Universal Robots PolyScope program: ur_comm_test_pal_depal_4times.urp

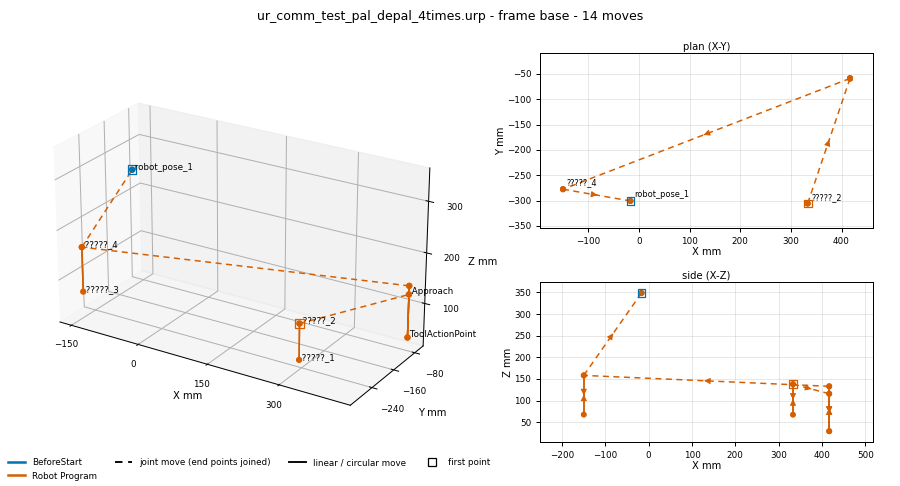
[picture p0: tool path of ur_comm_test_pal_depal_4times.urp in frame base, 14 of 14 moves have a stored position in this frame; points joined in program order, loops and branches not executed]
Program ur_comm_test_pal_depal_10times (installation=default directory=/programs/usbdisk/zivid-python-test/ur_comm_test_sample createdIn=5.5.1 lastSavedIn=5.21.0 robotSerialNumber=20195300395)
Calibrated DH parameters: a=[-0.000108, -0.14067, -0.21248, -0.000061, -0.000086, 0]; d=[0.151815, 81.30975, -77.69219, -3.486516, 0.085386, 0.091974]; alpha=[1.569683, -0.002449, 0.004563, 1.571204, -1.571811, 0]; deltaTheta=[0, -0.955759, 1.033289, -0.077525, 0.000001, 0]
InitVariablesNode variables(variable(name=Pallet_1_cnt, expression=1), variable(name=Pallet_1_cnt_1, expression=1), variable(name=Pallet_1_lct, expression=1), variable(name=Pallet_1_lct_1, expression=1), variable(name=Pallet_1_lno, expression=1), variable(name=Pallet_1_lno_1, expression=1), variable(name=Pallet_1_sep, expression=False), variable(name=Pallet_1_sep_1, expression=False), variable(name=Pallet_1_tct, expression=1), variable(name=Pallet_1_tct_1, expression=1), variable(name=qNearApproach, expression=[0,0,0,0,0,0]), variable(name=qNearApproach_1, expression=[0,0,0,0,0,0]))
BeforeStart
  Set DigitalOutput pin=conveyor_on; digitalValue=1
  count := 0
  URCap 2FG 놓기 (OnRobot, OnRobot A/S) dataModel(twofg.external-grip.target-width=0.03670000076293945, twofg.internal-grip.target-width=0.05070000076293945)
  MoveJ speed 15 deg/s, acceleration 15 deg/s^2 (useActiveTCP=true optimoveEnabled=true optiMoveSpeed=1 optiMoveAcceleration=1) feature=Base
    Waypoint robot_pose_1: TCP in base x=-16.534 y=-300.847 z=348.638 mm, rx=2.6839 ry=0.1063 rz=-0.0079 rad; joints [-46.382, -62.621, -71.979, -115.359, 73.035, -143.967] deg; TCP offset x=-7.625 y=23.932 z=143.735 mm, rx=0 ry=0 rz=0 rad
  Script: write_output_integer_register(24,count)
  Script: write_output_boolean_register(64,False)
Robot Program (runOnlyOnce=false)
  Wait Condition expression=read_input_boolean_register(125)
  count := count+1
  Script: write_output_integer_register(24,count)
  Script: write_output_boolean_register(64,True)
  Script: read_input_boolean_register(125)
  Loop Counting (count=4) loopVariable(name=루프_1)
    Loop Counting (count=6) loopVariable(name=루프_2)
      MoveJ speed 60 deg/s, acceleration 80 deg/s^2 (useActiveTCP=true optimoveEnabled=true optiMoveSpeed=1 optiMoveAcceleration=1) feature=Base
        Waypoint 웨이포인트_2: TCP in base x=333.162 y=-305.802 z=138.045 mm, rx=2.2214 ry=2.2214 rz=0 rad; joints [-26.216, -117.027, -61.814, -91.097, 90.185, -206.198] deg
      MoveL speed 250 mm/s, acceleration 1200 mm/s^2 (useActiveTCP=true optimoveEnabled=true optiMoveSpeed=1 optiMoveAcceleration=1) feature=Base
        Waypoint 웨이포인트_1: TCP in base x=333.162 y=-305.802 z=67.503 mm, rx=2.2214 ry=2.2214 rz=0 rad; joints [-26.24, -119.399, -77.36, -73.18, 90.18, -206.146] deg
        URCap 2FG 그립 (OnRobot, OnRobot A/S) dataModel(twofg.external-grip.target-width=0.02370000076293945, twofg.internal-grip.target-width=0.03770000076293945)
        Waypoint 웨이포인트_2: TCP in base x=333.162 y=-305.802 z=138.045 mm, rx=2.2214 ry=2.2214 rz=0 rad; joints [-26.216, -117.027, -61.814, -91.097, 90.185, -206.198] deg
      URCap 팔레타이징 (polyscope-pallet-impl, Universal Robots) dataModel(palletFeature=Base, isPalletizing=true, Variable(key=referencePoint, variable(featureName=referencePoint)), Variable(key=separatorPoint, variable(featureName=separatorPoint)), Variable(key=qNearApproach, variable(name=qNearApproach, initializeExpression=[0,0,0,0,0,0])), Variable(key=name, variable(name=Pallet_1)), Variable(key=globalCountingVariable, variable(name=Pallet_1_cnt, initializeExpression=1)), Variable(key=layerNumberVariable, variable(name=Pallet_1_lno, initializeExpression=1)), Variable(key=layerCountingVariable, variable(name=Pallet_1_lct, initializeExpression=1)), Variable(key=handleSeparatorVariable, variable(name=Pallet_1_sep, initializeExpression=False)), Variable(key=totalCountVariable, variable(name=Pallet_1_tct, initializeExpression=1)), Length(key=objectHeight value=0.03 unit=M)); state(isChildrenLocked=true)
        URCap 패턴 (polyscope-pallet-impl, Universal Robots) state(isChildrenLocked=true)
          URCap 패턴 (polyscope-pallet-impl, Universal Robots) dataModel(UUID=d919b560-e99a-480d-bc1f-cb570735da14, patternType=GRID, rows=3, columns=2, Variable(key=nameVariable, variable(name=Grid_Pattern_1))); state(isChildrenLocked=true)
            URCap 아이템 (polyscope-pallet-impl, Universal Robots) dataModel(UUID=ee1cad20-2e71-4b8d-ab70-a290e76e5d6c, patternType=GRID, index=0, calibrationDeltaTheta=[6.716763317901001E-8, -0.9557590612475653, 1.0332894801482315, -0.07752547289049558, 5.674308259095984E-7, -2.281062283008531E-7], calibrationA=[-1.0844059639211092E-4, -0.14067031953614179, -0.21248043873134673, -6.078177536491715E-5, -8.613979399887485E-5, 0.0], calibrationD=[0.15181475343250603, 81.30975015896925, -77.6921895952701, -3.486515920890218, 0.08538604408418736, 0.09197393797432639], calibrationAlpha=[1.569682990986815, -0.0024489725605047743, 0.004563020512108627, 1.571204384472482, -1.5718110539936228, 0.0], calibrationJointChecksum=[-1321669567, -1322594988, 822688479, -1328072335, -1327094287, -1329556568], calibrationStatus=2, calibrationValidChecksum=true, baseToFeature=[0.0, 0.0, 0.0, 0.0, 0.0, 0.0], TCPOffset=[-0.00762820289468219, 0.0239501142926695, 0.14372303756847724, -4.3315942804722315E-5, 7.042533500568108E-6, 2.3758754532917458E-5], Variable(key=variable, variable(name=CornerItem_1)), JointPositions(key=jointpositions, JointPosition(key=[1], Angle(key=pos value=0.230122 unit=RAD)), JointPosition(key=[2], Angle(key=pos value=-2.124559 unit=RAD)), JointPosition(key=[3], Angle(key=pos value=-1.476286 unit=RAD)), JointPosition(key=[4], Angle(key=pos value=-1.110532 unit=RAD)), JointPosition(key=[5], Angle(key=pos value=1.5737 unit=RAD)), JointPosition(key=[6], Angle(key=pos value=-1.360397 unit=RAD))))
            URCap 아이템 (polyscope-pallet-impl, Universal Robots) dataModel(UUID=2ec53ba5-ed44-4377-a54f-87662cf6edc9, patternType=GRID, index=1, calibrationDeltaTheta=[6.716763317901001E-8, -0.9557590612475653, 1.0332894801482315, -0.07752547289049558, 5.674308259095984E-7, -2.281062283008531E-7], calibrationA=[-1.0844059639211092E-4, -0.14067031953614179, -0.21248043873134673, -6.078177536491715E-5, -8.613979399887485E-5, 0.0], calibrationD=[0.15181475343250603, 81.30975015896925, -77.6921895952701, -3.486515920890218, 0.08538604408418736, 0.09197393797432639], calibrationAlpha=[1.569682990986815, -0.0024489725605047743, 0.004563020512108627, 1.571204384472482, -1.5718110539936228, 0.0], calibrationJointChecksum=[-1321669567, -1322594988, 822688479, -1328072335, -1327094287, -1329556568], calibrationStatus=2, calibrationValidChecksum=true, baseToFeature=[0.0, 0.0, 0.0, 0.0, 0.0, 0.0], TCPOffset=[-0.007627364228596889, 0.023926276031487913, 0.1437254493979939, 1.6298927572986975E-5, -1.936015947561922E-6, -2.0279970492899247E-5], Variable(key=variable, variable(name=CornerItem_2)), JointPositions(key=jointpositions, JointPosition(key=[1], Angle(key=pos value=0.32864 unit=RAD)), JointPosition(key=[2], Angle(key=pos value=-1.666236 unit=RAD)), JointPosition(key=[3], Angle(key=pos value=-2.130058 unit=RAD)), JointPosition(key=[4], Angle(key=pos value=-0.915088 unit=RAD)), JointPosition(key=[5], Angle(key=pos value=1.573564 unit=RAD)), JointPosition(key=[6], Angle(key=pos value=-1.259999 unit=RAD))))
            URCap 아이템 (polyscope-pallet-impl, Universal Robots) dataModel(UUID=892b0312-8469-4b11-924f-1544095aac69, patternType=GRID, index=2, calibrationDeltaTheta=[6.716763317901001E-8, -0.9557590612475653, 1.0332894801482315, -0.07752547289049558, 5.674308259095984E-7, -2.281062283008531E-7], calibrationA=[-1.0844059639211092E-4, -0.14067031953614179, -0.21248043873134673, -6.078177536491715E-5, -8.613979399887485E-5, 0.0], calibrationD=[0.15181475343250603, 81.30975015896925, -77.6921895952701, -3.486515920890218, 0.08538604408418736, 0.09197393797432639], calibrationAlpha=[1.569682990986815, -0.0024489725605047743, 0.004563020512108627, 1.571204384472482, -1.5718110539936228, 0.0], calibrationJointChecksum=[-1321669567, -1322594988, 822688479, -1328072335, -1327094287, -1329556568], calibrationStatus=2, calibrationValidChecksum=true, baseToFeature=[0.0, 0.0, 0.0, 0.0, 0.0, 0.0], TCPOffset=[-0.007639878420080737, 0.023943869668825668, 0.14373765785164358, -1.943663654326589E-5, -1.5468052752266034E-5, 3.456527941839842E-6], Variable(key=variable, variable(name=CornerItem_3)), JointPositions(key=jointpositions, JointPosition(key=[1], Angle(key=pos value=0.118809 unit=RAD)), JointPosition(key=[2], Angle(key=pos value=-1.718406 unit=RAD)), JointPosition(key=[3], Angle(key=pos value=-2.068775 unit=RAD)), JointPosition(key=[4], Angle(key=pos value=-0.924192 unit=RAD)), JointPosition(key=[5], Angle(key=pos value=1.573526 unit=RAD)), JointPosition(key=[6], Angle(key=pos value=-1.469977 unit=RAD))))
            URCap 아이템 (polyscope-pallet-impl, Universal Robots) dataModel(UUID=cf353ae9-dbdd-4e16-bdff-710f563f51b7, patternType=GRID, index=3, calibrationDeltaTheta=[6.716763317901001E-8, -0.9557590612475653, 1.0332894801482315, -0.07752547289049558, 5.674308259095984E-7, -2.281062283008531E-7], calibrationA=[-1.0844059639211092E-4, -0.14067031953614179, -0.21248043873134673, -6.078177536491715E-5, -8.613979399887485E-5, 0.0], calibrationD=[0.15181475343250603, 81.30975015896925, -77.6921895952701, -3.486515920890218, 0.08538604408418736, 0.09197393797432639], calibrationAlpha=[1.569682990986815, -0.0024489725605047743, 0.004563020512108627, 1.571204384472482, -1.5718110539936228, 0.0], calibrationJointChecksum=[-1321669567, -1322594988, 822688479, -1328072335, -1327094287, -1329556568], calibrationStatus=2, calibrationValidChecksum=true, baseToFeature=[0.0, 0.0, 0.0, 0.0, 0.0, 0.0], TCPOffset=[-0.0076283249516490015, 0.02393296756205482, 0.14376242105826337, -1.8085091406019513E-5, -4.76246665041877E-5, 1.1126998149954308E-5], Variable(key=variable, variable(name=CornerItem_4)), JointPositions(key=jointpositions, JointPosition(key=[1], Angle(key=pos value=0.080239 unit=RAD)), JointPosition(key=[2], Angle(key=pos value=-2.155316 unit=RAD)), JointPosition(key=[3], Angle(key=pos value=-1.42445 unit=RAD)), JointPosition(key=[4], Angle(key=pos value=-1.131606 unit=RAD)), JointPosition(key=[5], Angle(key=pos value=1.573688 unit=RAD)), JointPosition(key=[6], Angle(key=pos value=-1.510421 unit=RAD))))
        URCap 레이어 (polyscope-pallet-impl, Universal Robots) dataModel(separators=[false], selectedPatterns=[d919b560-e99a-480d-bc1f-cb570735da14])
        URCap 각각의 아이템 (polyscope-pallet-impl, Universal Robots) dataModel(selectedPattern=d919b560-e99a-480d-bc1f-cb570735da14, selectedPosition=ee1cad20-2e71-4b8d-ab70-a290e76e5d6c, Approach_calibrationDeltaTheta=[6.716763317901001E-8, -0.9557590612475653, 1.0332894801482315, -0.07752547289049558, 5.674308259095984E-7, -2.281062283008531E-7], Approach_calibrationA=[-1.0844059639211092E-4, -0.14067031953614179, -0.21248043873134673, -6.078177536491715E-5, -8.613979399887485E-5, 0.0], Approach_calibrationD=[0.15181475343250603, 81.30975015896925, -77.6921895952701, -3.486515920890218, 0.08538604408418736, 0.09197393797432639], Approach_calibrationAlpha=[1.569682990986815, -0.0024489725605047743, 0.004563020512108627, 1.571204384472482, -1.5718110539936228, 0.0], Approach_calibrationJointChecksum=[-1321669567, -1322594988, 822688479, -1328072335, -1327094287, -1329556568], Approach_calibrationStatus=2, Approach_calibrationValidChecksum=true, Approach_baseToFeature=[0.0, 0.0, 0.0, 0.0, 0.0, 0.0], Approach_TCPOffset=[-0.0076294742125221915, 0.02392315779155893, 0.14376079906325706, 2.9702410288334196E-5, -6.399436710385144E-5, -4.55675022656733E-5], Exit_calibrationDeltaTheta=[6.716763317901001E-8, -0.9557590612475653, 1.0332894801482315, -0.07752547289049558, 5.674308259095984E-7, -2.281062283008531E-7], Exit_calibrationA=[-1.0844059639211092E-4, -0.14067031953614179, -0.21248043873134673, -6.078177536491715E-5, -8.613979399887485E-5, 0.0], Exit_calibrationD=[0.15181475343250603, 81.30975015896925, -77.6921895952701, -3.486515920890218, 0.08538604408418736, 0.09197393797432639], Exit_calibrationAlpha=[1.569682990986815, -0.0024489725605047743, 0.004563020512108627, 1.571204384472482, -1.5718110539936228, 0.0], Exit_calibrationJointChecksum=[-1321669567, -1322594988, 822688479, -1328072335, -1327094287, -1329556568], Exit_calibrationStatus=2, Exit_calibrationValidChecksum=true, Exit_baseToFeature=[0.0, 0.0, 0.0, 0.0, 0.0, 0.0], Exit_TCPOffset=[-0.007615351300449602, 0.02389728385555888, 0.14374352147036207, 2.5680027780448787E-5, -3.149176289617292E-6, -3.7337634040478105E-5], currentWizardState=LANDING, Pose(key=refBaseToFeature, Position(key=posePosition, Length(key=X value=0 unit=M), Length(key=Y value=0 unit=M), Length(key=Z value=0 unit=M)), Rotation(key=poseRotation, Angle(key=RX value=0 unit=RAD), Angle(key=RY value=0 unit=RAD), Angle(key=RZ value=0 unit=RAD))), Pose(key=refPose, Position(key=posePosition, Length(key=X value=0.416803 unit=M), Length(key=Y value=-0.059002 unit=M), Length(key=Z value=0.029418 unit=M)), Rotation(key=poseRotation, Angle(key=RX value=3.14136 unit=RAD), Angle(key=RY value=0.034493 unit=RAD), Angle(key=RZ value=0.000012 unit=RAD))), JointPositions(key=Approach_jointpositions, JointPosition(key=[1], Angle(key=pos value=0.23048 unit=RAD)), JointPosition(key=[2], Angle(key=pos value=-2.025888 unit=RAD)), JointPosition(key=[3], Angle(key=pos value=-1.207737 unit=RAD)), JointPosition(key=[4], Angle(key=pos value=-1.477755 unit=RAD)), JointPosition(key=[5], Angle(key=pos value=1.574011 unit=RAD)), JointPosition(key=[6], Angle(key=pos value=-1.361408 unit=RAD))), JointPositions(key=Exit_jointpositions, JointPosition(key=[1], Angle(key=pos value=0.2306 unit=RAD)), JointPosition(key=[2], Angle(key=pos value=-2.021999 unit=RAD)), JointPosition(key=[3], Angle(key=pos value=-1.133203 unit=RAD)), JointPosition(key=[4], Angle(key=pos value=-1.556178 unit=RAD)), JointPosition(key=[5], Angle(key=pos value=1.574003 unit=RAD)), JointPosition(key=[6], Angle(key=pos value=-1.361636 unit=RAD))))
          URCap 생성된 이동 (polyscope-pallet-impl, Universal Robots) state(isChildrenLocked=true)
            MoveJ speed 60 deg/s, acceleration 80 deg/s^2 (useActiveTCP=true optimoveEnabled=true optiMoveSpeed=1 optiMoveAcceleration=1) feature=referencePoint
              Waypoint Approach: TCP in base x=416.798 y=-58.994 z=115.935 mm, rx=3.1414 ry=0.0346 rz=-0.0001 rad; joints [13.206, -116.075, -69.198, -84.669, 90.184, -78.003] deg; TCP offset x=-7.629 y=23.923 z=143.761 mm, rx=0 ry=-0.0001 rz=0 rad; feature pose in base x=416.803 y=-59.002 z=29.418 mm, rx=3.1414 ry=0.0345 rz=0 rad
            MoveL speed 250 mm/s, acceleration 1200 mm/s^2 (useActiveTCP=true optimoveEnabled=true optiMoveSpeed=1 optiMoveAcceleration=1) feature(featureName=referencePoint)
              Waypoint ToolActionPoint: TCP in base x=416.803 y=-59.002 z=29.418 mm, rx=3.1414 ry=0.0345 rz=0 rad; joints [13.185, -121.728, -84.585, -63.629, 90.166, -77.945] deg; TCP offset x=-7.628 y=23.95 z=143.723 mm, rx=0 ry=0 rz=0 rad
            Folder Tool action
              URCap 2FG 놓기 (OnRobot, OnRobot A/S) dataModel(twofg.external-grip.target-width=0.03670000076293945, twofg.internal-grip.target-width=0.05070000076293945)
            MoveL speed 250 mm/s, acceleration 1200 mm/s^2 (useActiveTCP=true optimoveEnabled=true optiMoveSpeed=1 optiMoveAcceleration=1) feature(featureName=referencePoint)
              Waypoint Exit: TCP in base x=416.812 y=-58.968 z=133.052 mm, rx=3.1414 ry=0.0346 rz=0 rad; joints [13.212, -115.852, -64.928, -89.162, 90.184, -78.016] deg; TCP offset x=-7.615 y=23.897 z=143.744 mm, rx=0 ry=0 rz=0 rad
    Loop Counting (count=6) loopVariable(name=루프_3)
      URCap 팔레타이징 (polyscope-pallet-impl, Universal Robots) dataModel(palletFeature=Base, isPalletizing=false, Length(key=objectHeight value=0.03 unit=M), Variable(key=referencePoint, variable(featureName=referencePoin_1)), Variable(key=separatorPoint, variable(featureName=separatorPoin_1)), Variable(key=qNearApproach, variable(name=qNearApproach_1, initializeExpression=[0,0,0,0,0,0])), Variable(key=name, variable(name=Pallet_2)), Variable(key=globalCountingVariable, variable(name=Pallet_1_cnt_1, initializeExpression=1)), Variable(key=layerCountingVariable, variable(name=Pallet_1_lct_1, initializeExpression=1)), Variable(key=layerNumberVariable, variable(name=Pallet_1_lno_1, initializeExpression=1)), Variable(key=handleSeparatorVariable, variable(name=Pallet_1_sep_1, initializeExpression=False)), Variable(key=totalCountVariable, variable(name=Pallet_1_tct_1, initializeExpression=1))); state(isChildrenLocked=true)
        URCap 패턴 (polyscope-pallet-impl, Universal Robots) state(isChildrenLocked=true)
          URCap 패턴 (polyscope-pallet-impl, Universal Robots) dataModel(UUID=d919b560-e99a-480d-bc1f-cb570735da14, patternType=GRID, rows=3, columns=2, Variable(key=nameVariable, variable(name=Grid_Pattern_2))); state(isChildrenLocked=true)
            URCap 아이템 (polyscope-pallet-impl, Universal Robots) dataModel(UUID=ee1cad20-2e71-4b8d-ab70-a290e76e5d6c, patternType=GRID, index=0, calibrationDeltaTheta=[6.716763317901001E-8, -0.9557590612475653, 1.0332894801482315, -0.07752547289049558, 5.674308259095984E-7, -2.281062283008531E-7], calibrationA=[-1.0844059639211092E-4, -0.14067031953614179, -0.21248043873134673, -6.078177536491715E-5, -8.613979399887485E-5, 0.0], calibrationD=[0.15181475343250603, 81.30975015896925, -77.6921895952701, -3.486515920890218, 0.08538604408418736, 0.09197393797432639], calibrationAlpha=[1.569682990986815, -0.0024489725605047743, 0.004563020512108627, 1.571204384472482, -1.5718110539936228, 0.0], calibrationJointChecksum=[-1321669567, -1322594988, 822688479, -1328072335, -1327094287, -1329556568], calibrationStatus=2, calibrationValidChecksum=true, baseToFeature=[0.0, 0.0, 0.0, 0.0, 0.0, 0.0], TCPOffset=[-0.00762820289468219, 0.0239501142926695, 0.14372303756847724, -4.3315942804722315E-5, 7.042533500568108E-6, 2.3758754532917458E-5], JointPositions(key=jointpositions, JointPosition(key=[1], Angle(key=pos value=0.230122 unit=RAD)), JointPosition(key=[2], Angle(key=pos value=-2.124559 unit=RAD)), JointPosition(key=[3], Angle(key=pos value=-1.476286 unit=RAD)), JointPosition(key=[4], Angle(key=pos value=-1.110532 unit=RAD)), JointPosition(key=[5], Angle(key=pos value=1.5737 unit=RAD)), JointPosition(key=[6], Angle(key=pos value=-1.360397 unit=RAD))), Variable(key=variable, variable(name=CornerItem_5)))
            URCap 아이템 (polyscope-pallet-impl, Universal Robots) dataModel(UUID=2ec53ba5-ed44-4377-a54f-87662cf6edc9, patternType=GRID, index=1, calibrationDeltaTheta=[6.716763317901001E-8, -0.9557590612475653, 1.0332894801482315, -0.07752547289049558, 5.674308259095984E-7, -2.281062283008531E-7], calibrationA=[-1.0844059639211092E-4, -0.14067031953614179, -0.21248043873134673, -6.078177536491715E-5, -8.613979399887485E-5, 0.0], calibrationD=[0.15181475343250603, 81.30975015896925, -77.6921895952701, -3.486515920890218, 0.08538604408418736, 0.09197393797432639], calibrationAlpha=[1.569682990986815, -0.0024489725605047743, 0.004563020512108627, 1.571204384472482, -1.5718110539936228, 0.0], calibrationJointChecksum=[-1321669567, -1322594988, 822688479, -1328072335, -1327094287, -1329556568], calibrationStatus=2, calibrationValidChecksum=true, baseToFeature=[0.0, 0.0, 0.0, 0.0, 0.0, 0.0], TCPOffset=[-0.007627364228596889, 0.023926276031487913, 0.1437254493979939, 1.6298927572986975E-5, -1.936015947561922E-6, -2.0279970492899247E-5], JointPositions(key=jointpositions, JointPosition(key=[1], Angle(key=pos value=0.32864 unit=RAD)), JointPosition(key=[2], Angle(key=pos value=-1.666236 unit=RAD)), JointPosition(key=[3], Angle(key=pos value=-2.130058 unit=RAD)), JointPosition(key=[4], Angle(key=pos value=-0.915088 unit=RAD)), JointPosition(key=[5], Angle(key=pos value=1.573564 unit=RAD)), JointPosition(key=[6], Angle(key=pos value=-1.259999 unit=RAD))), Variable(key=variable, variable(name=CornerItem_6)))
            URCap 아이템 (polyscope-pallet-impl, Universal Robots) dataModel(UUID=892b0312-8469-4b11-924f-1544095aac69, patternType=GRID, index=2, calibrationDeltaTheta=[6.716763317901001E-8, -0.9557590612475653, 1.0332894801482315, -0.07752547289049558, 5.674308259095984E-7, -2.281062283008531E-7], calibrationA=[-1.0844059639211092E-4, -0.14067031953614179, -0.21248043873134673, -6.078177536491715E-5, -8.613979399887485E-5, 0.0], calibrationD=[0.15181475343250603, 81.30975015896925, -77.6921895952701, -3.486515920890218, 0.08538604408418736, 0.09197393797432639], calibrationAlpha=[1.569682990986815, -0.0024489725605047743, 0.004563020512108627, 1.571204384472482, -1.5718110539936228, 0.0], calibrationJointChecksum=[-1321669567, -1322594988, 822688479, -1328072335, -1327094287, -1329556568], calibrationStatus=2, calibrationValidChecksum=true, baseToFeature=[0.0, 0.0, 0.0, 0.0, 0.0, 0.0], TCPOffset=[-0.007639878420080737, 0.023943869668825668, 0.14373765785164358, -1.943663654326589E-5, -1.5468052752266034E-5, 3.456527941839842E-6], JointPositions(key=jointpositions, JointPosition(key=[1], Angle(key=pos value=0.118809 unit=RAD)), JointPosition(key=[2], Angle(key=pos value=-1.718406 unit=RAD)), JointPosition(key=[3], Angle(key=pos value=-2.068775 unit=RAD)), JointPosition(key=[4], Angle(key=pos value=-0.924192 unit=RAD)), JointPosition(key=[5], Angle(key=pos value=1.573526 unit=RAD)), JointPosition(key=[6], Angle(key=pos value=-1.469977 unit=RAD))), Variable(key=variable, variable(name=CornerItem_7)))
            URCap 아이템 (polyscope-pallet-impl, Universal Robots) dataModel(UUID=cf353ae9-dbdd-4e16-bdff-710f563f51b7, patternType=GRID, index=3, calibrationDeltaTheta=[6.716763317901001E-8, -0.9557590612475653, 1.0332894801482315, -0.07752547289049558, 5.674308259095984E-7, -2.281062283008531E-7], calibrationA=[-1.0844059639211092E-4, -0.14067031953614179, -0.21248043873134673, -6.078177536491715E-5, -8.613979399887485E-5, 0.0], calibrationD=[0.15181475343250603, 81.30975015896925, -77.6921895952701, -3.486515920890218, 0.08538604408418736, 0.09197393797432639], calibrationAlpha=[1.569682990986815, -0.0024489725605047743, 0.004563020512108627, 1.571204384472482, -1.5718110539936228, 0.0], calibrationJointChecksum=[-1321669567, -1322594988, 822688479, -1328072335, -1327094287, -1329556568], calibrationStatus=2, calibrationValidChecksum=true, baseToFeature=[0.0, 0.0, 0.0, 0.0, 0.0, 0.0], TCPOffset=[-0.0076283249516490015, 0.02393296756205482, 0.14376242105826337, -1.8085091406019513E-5, -4.76246665041877E-5, 1.1126998149954308E-5], JointPositions(key=jointpositions, JointPosition(key=[1], Angle(key=pos value=0.080239 unit=RAD)), JointPosition(key=[2], Angle(key=pos value=-2.155316 unit=RAD)), JointPosition(key=[3], Angle(key=pos value=-1.42445 unit=RAD)), JointPosition(key=[4], Angle(key=pos value=-1.131606 unit=RAD)), JointPosition(key=[5], Angle(key=pos value=1.573688 unit=RAD)), JointPosition(key=[6], Angle(key=pos value=-1.510421 unit=RAD))), Variable(key=variable, variable(name=CornerItem_8)))
        URCap 레이어 (polyscope-pallet-impl, Universal Robots) dataModel(separators=[false], selectedPatterns=[d919b560-e99a-480d-bc1f-cb570735da14])
        URCap 각각의 아이템 (polyscope-pallet-impl, Universal Robots) dataModel(selectedPattern=d919b560-e99a-480d-bc1f-cb570735da14, selectedPosition=ee1cad20-2e71-4b8d-ab70-a290e76e5d6c, Approach_calibrationDeltaTheta=[6.716763317901001E-8, -0.9557590612475653, 1.0332894801482315, -0.07752547289049558, 5.674308259095984E-7, -2.281062283008531E-7], Approach_calibrationA=[-1.0844059639211092E-4, -0.14067031953614179, -0.21248043873134673, -6.078177536491715E-5, -8.613979399887485E-5, 0.0], Approach_calibrationD=[0.15181475343250603, 81.30975015896925, -77.6921895952701, -3.486515920890218, 0.08538604408418736, 0.09197393797432639], Approach_calibrationAlpha=[1.569682990986815, -0.0024489725605047743, 0.004563020512108627, 1.571204384472482, -1.5718110539936228, 0.0], Approach_calibrationJointChecksum=[-1321669567, -1322594988, 822688479, -1328072335, -1327094287, -1329556568], Approach_calibrationStatus=2, Approach_calibrationValidChecksum=true, Approach_baseToFeature=[0.0, 0.0, 0.0, 0.0, 0.0, 0.0], Approach_TCPOffset=[-0.0076294742125221915, 0.02392315779155893, 0.14376079906325706, 2.9702410288334196E-5, -6.399436710385144E-5, -4.55675022656733E-5], Exit_calibrationDeltaTheta=[6.716763317901001E-8, -0.9557590612475653, 1.0332894801482315, -0.07752547289049558, 5.674308259095984E-7, -2.281062283008531E-7], Exit_calibrationA=[-1.0844059639211092E-4, -0.14067031953614179, -0.21248043873134673, -6.078177536491715E-5, -8.613979399887485E-5, 0.0], Exit_calibrationD=[0.15181475343250603, 81.30975015896925, -77.6921895952701, -3.486515920890218, 0.08538604408418736, 0.09197393797432639], Exit_calibrationAlpha=[1.569682990986815, -0.0024489725605047743, 0.004563020512108627, 1.571204384472482, -1.5718110539936228, 0.0], Exit_calibrationJointChecksum=[-1321669567, -1322594988, 822688479, -1328072335, -1327094287, -1329556568], Exit_calibrationStatus=2, Exit_calibrationValidChecksum=true, Exit_baseToFeature=[0.0, 0.0, 0.0, 0.0, 0.0, 0.0], Exit_TCPOffset=[-0.007615351300449602, 0.02389728385555888, 0.14374352147036207, 2.5680027780448787E-5, -3.149176289617292E-6, -3.7337634040478105E-5], currentWizardState=LANDING, Pose(key=refBaseToFeature, Position(key=posePosition, Length(key=X value=0 unit=M), Length(key=Y value=0 unit=M), Length(key=Z value=0 unit=M)), Rotation(key=poseRotation, Angle(key=RX value=0 unit=RAD), Angle(key=RY value=0 unit=RAD), Angle(key=RZ value=0 unit=RAD))), Pose(key=refPose, Position(key=posePosition, Length(key=X value=0.416803 unit=M), Length(key=Y value=-0.059002 unit=M), Length(key=Z value=0.029418 unit=M)), Rotation(key=poseRotation, Angle(key=RX value=3.14136 unit=RAD), Angle(key=RY value=0.034493 unit=RAD), Angle(key=RZ value=0.000012 unit=RAD))), JointPositions(key=Approach_jointpositions, JointPosition(key=[1], Angle(key=pos value=0.23048 unit=RAD)), JointPosition(key=[2], Angle(key=pos value=-2.025888 unit=RAD)), JointPosition(key=[3], Angle(key=pos value=-1.207737 unit=RAD)), JointPosition(key=[4], Angle(key=pos value=-1.477755 unit=RAD)), JointPosition(key=[5], Angle(key=pos value=1.574011 unit=RAD)), JointPosition(key=[6], Angle(key=pos value=-1.361408 unit=RAD))), JointPositions(key=Exit_jointpositions, JointPosition(key=[1], Angle(key=pos value=0.2306 unit=RAD)), JointPosition(key=[2], Angle(key=pos value=-2.021999 unit=RAD)), JointPosition(key=[3], Angle(key=pos value=-1.133203 unit=RAD)), JointPosition(key=[4], Angle(key=pos value=-1.556178 unit=RAD)), JointPosition(key=[5], Angle(key=pos value=1.574003 unit=RAD)), JointPosition(key=[6], Angle(key=pos value=-1.361636 unit=RAD))))
          URCap 생성된 이동 (polyscope-pallet-impl, Universal Robots) state(isChildrenLocked=true)
            MoveJ speed 60 deg/s, acceleration 80 deg/s^2 (useActiveTCP=true optimoveEnabled=true optiMoveSpeed=1 optiMoveAcceleration=1) feature=referencePoin_1
              Waypoint Approach: TCP in base x=416.798 y=-58.994 z=115.935 mm, rx=3.1414 ry=0.0346 rz=-0.0001 rad; joints [13.206, -116.075, -69.198, -84.669, 90.184, -78.003] deg; TCP offset x=-7.629 y=23.923 z=143.761 mm, rx=0 ry=-0.0001 rz=0 rad
            MoveL speed 250 mm/s, acceleration 1200 mm/s^2 (useActiveTCP=true optimoveEnabled=true optiMoveSpeed=1 optiMoveAcceleration=1) feature(featureName=referencePoin_1)
              Waypoint ToolActionPoint: TCP in base x=416.803 y=-59.002 z=29.418 mm, rx=3.1414 ry=0.0345 rz=0 rad; joints [13.185, -121.728, -84.585, -63.629, 90.166, -77.945] deg; TCP offset x=-7.628 y=23.95 z=143.723 mm, rx=0 ry=0 rz=0 rad
            Folder Tool action
              URCap 2FG 그립 (OnRobot, OnRobot A/S) dataModel(twofg.external-grip.target-width=0.02370000076293945, twofg.internal-grip.target-width=0.03770000076293945)
            MoveL speed 250 mm/s, acceleration 1200 mm/s^2 (useActiveTCP=true optimoveEnabled=true optiMoveSpeed=1 optiMoveAcceleration=1) feature(featureName=referencePoin_1)
              Waypoint Exit: TCP in base x=416.812 y=-58.968 z=133.052 mm, rx=3.1414 ry=0.0346 rz=0 rad; joints [13.212, -115.852, -64.928, -89.162, 90.184, -78.016] deg; TCP offset x=-7.615 y=23.897 z=143.744 mm, rx=0 ry=0 rz=0 rad
      MoveJ speed 60 deg/s, acceleration 80 deg/s^2 (useActiveTCP=true optimoveEnabled=true optiMoveSpeed=1 optiMoveAcceleration=1) feature=Base
        Waypoint 웨이포인트_4: TCP in base x=-149.78 y=-277.687 z=158.255 mm, rx=-2.191 ry=2.2515 rz=0 rad; joints [-89.108, -86.57, -93.896, -89.476, 90.215, -87.455] deg; TCP offset x=-7.625 y=23.932 z=143.735 mm, rx=0 ry=0 rz=0 rad
      MoveL speed 250 mm/s, acceleration 1200 mm/s^2 (useActiveTCP=true optimoveEnabled=true optiMoveSpeed=1 optiMoveAcceleration=1) feature=Base
        Waypoint 웨이포인트_3: TCP in base x=-149.78 y=-277.687 z=67.712 mm, rx=-2.191 ry=2.2515 rz=0 rad; joints [-89.143, -91.506, -114.239, -64.197, 90.191, -87.387] deg
        URCap 2FG 놓기 (OnRobot, OnRobot A/S) dataModel(twofg.external-grip.target-width=0.03670000076293945, twofg.internal-grip.target-width=0.05070000076293945)
        Waypoint 웨이포인트_4: TCP in base x=-149.78 y=-277.687 z=158.255 mm, rx=-2.191 ry=2.2515 rz=0 rad; joints [-89.108, -86.57, -93.896, -89.476, 90.215, -87.455] deg
    count := count+1
    Script: write_output_integer_register(24,count)
  Wait Sleep waitTime=0.5
  Script: write_output_integer_register(24,-1)
  MoveJ speed 15 deg/s, acceleration 15 deg/s^2 (useActiveTCP=true optimoveEnabled=true optiMoveSpeed=1 optiMoveAcceleration=1) feature=Base
    Waypoint robot_pose_1: TCP in base x=-16.534 y=-300.847 z=348.638 mm, rx=2.6839 ry=0.1063 rz=-0.0079 rad; joints [-46.382, -62.621, -71.979, -115.359, 73.035, -143.967] deg
  Set DigitalOutput pin=conveyor_on; digitalValue=0
  Halt
